Yaskawa INFORM job: SKRZYNIA_5440_90_STOPNI_20BR.JBI

/JOB
//NAME SKRZYNIA_5440_90_STOPNI_20BR
///FOLDERNAME 02-SKRZYNIE_JOBS
//POS
///NPOS 570,570,0,41,0,0
///TOOL 0
///POSTYPE PULSE
///PULSE
C00000=0,-52280,40443,0,6876,0
C00001=82314,-24956,17040,59626,-27382,6248
C00002=93910,-8625,17040,59626,-43355,6248
C00003=98846,-1061,-42166,80308,-57081,-16120
C00004=100452,6057,-48127,85711,-56704,-21322
C00005=95573,33077,-33257,84645,-64023,-26851
C00006=94102,33899,-31937,85246,-63371,-26689
C00007=95573,33077,-33257,84645,-64023,-26851
C00008=94862,31071,-36438,85313,-63677,-27192
C00009=95573,33077,-33257,84645,-64023,-26851
C00010=95263,33142,-33256,84677,-63995,-26850
C00011=95263,33142,-33256,84677,-63995,-26850
C00012=94017,33843,-32133,85187,-63445,-26710
C00013=95263,33142,-33256,84677,-63995,-26850
C00014=94657,31439,-35966,85248,-63701,-27141
C00015=95263,33142,-33256,84677,-63995,-26850
C00016=95260,33144,-33256,84678,-63995,-26850
C00017=95260,33144,-33256,84678,-63995,-26850
C00018=94022,33838,-32141,85183,-63448,-26711
C00019=95260,33144,-33256,84678,-63995,-26850
C00020=94618,31343,-36117,85281,-63684,-27157
C00021=95260,33144,-33256,84678,-63995,-26850
C00022=95258,25631,32269,66559,-75499,-2416
C00023=95258,25631,32269,66559,-75499,-2416
C00024=94181,26497,33533,66410,-74896,-2191
C00025=95658,30184,39035,66708,-78559,-2356
C00026=95217,30377,39331,66881,-79841,-2558
C00027=95258,25631,32269,66559,-75499,-2416
C00028=98811,21047,-15512,99242,-81394,-20987
C00029=98811,21047,-15512,99242,-81394,-20987
C00030=97775,21639,-14693,99563,-80753,-20993
C00031=98811,21047,-15512,99242,-81394,-20987
C00032=98206,18840,-18520,99489,-81124,-21211
C00033=98811,21047,-15512,99242,-81394,-20987
C00034=98765,34858,63506,90961,-74847,-417
C00035=98765,34858,63506,90961,-74847,-417
C00036=97741,35895,65220,90657,-74158,-246
C00037=98765,34858,63506,90961,-74847,-417
C00038=98337,32226,59232,91111,-74633,-884
C00039=98765,34858,63506,90961,-74847,-417
C00040=98728,21792,17445,103800,-78809,-12049
C00041=97232,27021,37502,101932,-75086,-7690
C00042=96358,27701,38514,101868,-74464,-7680
C00043=97232,27021,37502,101932,-75086,-7690
C00044=96733,24820,34282,102049,-74905,-7989
C00045=97232,27021,37502,101932,-75086,-7690
C00046=94428,854,16076,89248,-50738,-4740
C00047=88080,-20128,-3199,80943,-31244,-2335
C00048=48287,-44591,-17414,16172,-14532,25809
C00049=48287,-44591,-17414,16172,-14532,25809
C00050=86232,-22530,-5035,79517,-30097,-1713
C00051=97395,20012,29210,69700,-74457,-9077
C00052=97055,28839,36684,71776,-79389,-10554
C00053=97055,28839,36684,71776,-79389,-10554
C00054=96058,29646,37897,71666,-78799,-10362
C00055=97055,28839,36684,71776,-79389,-10554
C00056=96570,26659,33451,71832,-78911,-10777
C00057=97055,28839,36684,71776,-79389,-10554
C00058=99123,23256,18377,81563,-78104,3156
C00059=99123,23256,18377,81563,-78104,3156
C00060=98123,23909,19300,81582,-77442,3256
C00061=99123,23256,18377,81563,-78104,3156
C00062=98765,21723,16234,81638,-77830,3017
C00063=99123,23256,18377,81563,-78104,3156
C00064=99222,23346,17795,82202,-78388,4176
C00065=99222,23346,17795,82202,-78388,4176
C00066=98149,24045,18779,82229,-77677,4281
C00067=99222,23346,17795,82202,-78388,4176
C00068=98861,21801,15633,82278,-78114,4033
C00069=99222,23346,17795,82202,-78388,4176
C00070=101181,20053,13227,82362,-77850,3884
C00071=98477,12630,5837,99042,-72451,1602
C00072=98699,20516,16868,97574,-77073,2916
C00073=97285,21426,18123,97638,-76093,2915
C00074=98699,20516,16868,97574,-77073,2916
C00075=98338,19050,14867,97654,-76881,2766
C00076=98699,20516,16868,97574,-77073,2916
C00077=100004,19406,13931,91923,-76989,3541
C00078=99329,-2479,-35949,113241,-72472,-2557
C00079=60067,-64368,-72505,144806,-26050,-19168
C00080=60067,-50244,-32501,110603,-14199,-2207
C00081=63330,-26972,24478,18707,-56801,31483
C00082=87404,-10792,18065,42799,-49272,19535
C00083=97387,10585,22601,68146,-67072,4966
C00084=97468,27299,36957,71364,-78144,1860
C00085=96326,28190,38285,71210,-77468,2075
C00086=97482,27286,36940,71366,-78155,1858
C00087=97039,25308,34039,71414,-77723,1669
C00088=97482,27286,36940,71366,-78155,1858
C00089=99359,23449,25979,91431,-77368,-3620
C00090=98281,24164,26997,91405,-76622,-3568
C00091=99359,23449,25979,91431,-77368,-3620
C00092=98971,21749,23585,91505,-77132,-3802
C00093=99359,23449,25979,91431,-77368,-3620
C00094=96616,4564,7202,89178,-62130,-2525
C00095=94710,-18885,-12427,84555,-44606,134
C00096=42754,-66126,12236,-1301,3231,7194
C00097=0,-52280,40443,0,6876,0
C00098=0,-52280,40443,0,6876,0
C00099=48041,-29633,723,44271,-15597,-57965
C00100=48041,-29633,723,44271,-15597,-57965
C00101=55649,-15396,14646,74799,-19245,-69915
C00102=54283,-14162,15682,74499,-18354,-69938
C00103=56054,-13547,16209,75912,-19428,-70417
C00104=55649,-15396,14646,74799,-19245,-69915
C00105=51081,-17733,11598,53117,-16128,-61899
C00106=49703,-16390,12674,51759,-15261,-61403
C00107=50366,-16427,12642,52774,-15606,-61824
C00108=49536,-18455,11034,50297,-15435,-60714
C00109=50509,-19000,10610,51503,-15997,-61182
C00110=50873,-17966,11417,52677,-16048,-61710
C00111=49459,-16590,12517,51258,-15158,-61190
C00112=50592,-16429,12648,53120,-15720,-61960
C00113=50873,-17966,11417,52677,-16048,-61710
C00114=50703,-18403,11066,52155,-16024,-61477
C00115=50703,-18403,11066,52155,-16024,-61477
C00116=49026,-16768,12358,50435,-14971,-60844
C00117=50653,-16371,12680,53228,-15754,-62008
C00118=50703,-18403,11066,52155,-16024,-61477
C00119=50704,-18401,11069,52157,-16021,-61478
C00120=50704,-20525,5414,58956,-14779,-64789
C00121=49025,-18889,6668,57745,-13658,-64384
C00122=50799,-18420,7036,60610,-14610,-65581
C00123=50704,-20525,5414,58956,-14779,-64789
C00124=51005,-17995,11387,52847,-16122,-61778
C00125=51005,-17995,11387,52847,-16122,-61778
C00126=49564,-16598,12501,51417,-15218,-61257
C00127=50954,-16306,12737,53719,-15902,-62212
C00128=51005,-17995,11387,52847,-16122,-61778
C00129=51030,-17981,11395,52891,-16138,-61796
C00130=51030,-17981,11395,52891,-16138,-61796
C00131=49401,-16396,12662,51265,-15114,-61201
C00132=50908,-16047,12947,53789,-15850,-62250
C00133=51030,-17981,11395,52891,-16138,-61796
C00134=50945,-18019,11363,52741,-16103,-61737
C00135=50945,-16980,14081,49884,-16761,-60338
C00136=49117,-15186,15539,47848,-15653,-59576
C00137=50939,-14679,15960,50992,-16487,-60881
C00138=50945,-18019,11363,52741,-16103,-61737
C00139=50945,-18019,11363,52741,-16103,-61737
C00140=50945,-18556,9943,54337,-15776,-62517
C00141=48967,-16606,11493,52445,-14510,-61829
C00142=51083,-15952,12027,56053,-15559,-63336
C00143=50945,-18556,9943,54337,-15776,-62517
C00144=50945,-18019,11363,52741,-16103,-61737
C00145=51350,-15183,18375,46705,-17991,-58719
C00146=49319,-13187,20053,44263,-16830,-57796
C00147=51236,-12618,20544,47529,-17647,-59142
C00148=51350,-15183,18375,46705,-17991,-58719
C00149=50028,-23690,-6096,22921,-31075,-54538
C00150=50670,-23735,-6923,24003,-30760,-55076
C00151=48518,-21492,-5254,21861,-29696,-54082
C00152=50138,-21068,-4928,23831,-30039,-55022
C00153=50670,-23735,-6923,24003,-30760,-55076
C00154=49763,-24225,-29961,22080,-30065,-59113
C00155=49763,-24225,-29961,22080,-30065,-59113
C00156=47727,-21550,-27874,20313,-29013,-58119
C00157=49271,-21042,-27466,22016,-29310,-59069
C00158=49763,-24225,-29961,22080,-30065,-59113
C00159=50713,-12366,-58367,41124,-17813,-74400
C00160=50713,-12366,-58367,41124,-17813,-74400
C00161=48934,-9522,-55687,39981,-16902,-73526
C00162=50242,-8975,-55157,41389,-17374,-74448
C00163=50713,-12366,-58367,41124,-17813,-74400
C00164=50713,-12366,-58367,41124,-17813,-74400
C00165=50713,-12366,-58367,41124,-17813,-74400
C00166=48934,-9522,-55687,39981,-16902,-73526
C00167=50242,-8975,-55157,41389,-17374,-74448
C00168=50713,-12366,-58367,41124,-17813,-74400
C00169=49763,-25421,-36239,24565,-26935,-60445
C00170=43547,-31626,-19626,5157,-49140,-52118
C00171=40154,-51179,-915,24203,-8234,-36524
C00172=0,-52280,40443,0,6876,0
C00173=0,-52280,40443,0,6876,0
C00174=2117,-50103,-33543,4117,45077,-85249
C00175=-26439,-48928,-33543,4117,-52362,-85249
C00176=-1453,-29933,-32011,46693,-66666,-90474
C00177=24798,-19255,-10490,69050,-85424,-90395
C00178=18386,-22028,-12683,68302,-81515,-89477
///LIMIT ON
C00179=9843,-31743,-57176,61611,-65235,-99401
C00180=-39603,-23393,-71448,91573,-31907,-107123
C00181=-35705,5077,-63140,100511,-35979,-118164
C00182=-33789,12193,-59259,102607,-37482,-119984
C00183=-34998,13124,-58049,103267,-36945,-119997
C00184=-34401,14597,-56112,102586,-37131,-119778
C00185=-34998,13124,-58049,103267,-36945,-119997
C00186=-36388,13885,-57049,104079,-36338,-120048
C00187=-34998,13124,-58049,103267,-36945,-119997
C00188=-34008,-7969,-75285,118537,-50852,-116988
C00189=-26318,8527,-57077,128458,-81874,-108613
///LIMIT OFF
C00190=-23139,-1795,-12064,73373,-53703,-87448
C00191=-27830,-667,-10848,73187,-50621,-86997
C00192=-27373,916,-9115,73207,-50922,-87041
C00193=-27830,-667,-10848,73187,-50621,-86997
C00194=-28901,-207,-10348,73132,-49918,-86888
C00195=-27830,-667,-10848,73187,-50621,-86997
C00196=-37166,8347,13175,41366,-53536,-76331
C00197=-37403,7707,12401,41298,-53388,-76282
C00198=-36830,9273,14303,41455,-53750,-76396
C00199=-37403,7707,12401,41298,-53388,-76282
C00200=-38235,8246,13056,40951,-53040,-76025
C00201=-37403,7707,12401,41298,-53388,-76282
C00202=-30063,5992,18551,55847,-56234,-77619
C00203=-30754,7414,19761,55747,-55713,-77591
C00204=-30376,8670,21285,55817,-55984,-77619
C00205=-30754,7414,19761,55747,-55713,-77591
C00206=-31265,7672,20073,55566,-55435,-77478
C00207=-30085,6037,18588,55845,-56218,-77619
C00208=-25385,-1715,-9470,94765,-53990,-89712
C00209=-25885,-764,-8323,94779,-53645,-89697
C00210=-25564,418,-7032,94741,-53861,-89683
C00211=-25885,-764,-8323,94779,-53645,-89697
C00212=-26741,-428,-7957,94890,-53068,-89741
C00213=-25421,-1648,-9389,94767,-53966,-89710
C00214=-17789,-39335,-40320,90232,-41783,-86178
C00215=-25885,-761,-8324,94780,-53645,-89696
C00216=-25885,-761,-8324,94780,-53645,-89696
C00217=-25612,239,-7230,94748,-53828,-89684
C00218=-25885,-761,-8324,94780,-53645,-89696
C00219=-26712,-436,-7972,94885,-53087,-89742
C00220=-25885,-761,-8324,94780,-53645,-89696
C00221=-26038,-1317,-8919,94796,-53541,-89701
C00222=-18430,-29121,-33898,93348,-44706,-88207
C00223=-3209,-48313,-44409,84985,-37126,-83197
C00224=-3617,-53456,-46461,81793,-37023,-81323
C00225=-28991,-22310,-29554,94749,-46554,-89251
C00226=-30664,-6343,-14094,96248,-45630,-90223
C00227=-30664,-6343,-14094,96248,-45630,-90223
C00228=-30207,-5031,-12762,96238,-45949,-90236
C00229=-30664,-6343,-14094,96248,-45630,-90223
C00230=-31510,-5971,-13720,96406,-45066,-90297
C00231=-29506,-9179,-17232,96085,-46411,-90159
C00232=-30003,-8487,-16482,96169,-46079,-90194
C00233=-30881,-6301,-14053,96286,-45485,-90239
C00234=-30407,-4956,-12684,96275,-45813,-90252
C00235=-30881,-6301,-14053,96286,-45485,-90239
C00236=-31646,-5963,-13712,96429,-44974,-90305
C00237=-29893,-8752,-16772,96152,-46152,-90188
C00238=-30350,-7636,-15544,96220,-45845,-90215
C00239=-30881,-6301,-14053,96286,-45485,-90239
C00240=-30396,-4924,-12652,96275,-45822,-90251
C00241=-30881,-6301,-14053,96286,-45485,-90239
C00242=-31665,-5954,-13703,96434,-44961,-90308
C00243=-29959,-8593,-16598,96162,-46108,-90192
C00244=-26558,-19284,-27675,95285,-48332,-89713
C00245=-5136,-57382,-50746,80999,-31115,-81799
C00246=-5136,-57382,-50746,80999,-31115,-81799
C00247=-22762,-12288,-20025,94001,-55646,-89200
C00248=-24763,-3131,-11201,94769,-54426,-89746
C00249=-26203,-419,-7954,94818,-53430,-89712
C00250=-25939,548,-6896,94784,-53609,-89698
C00251=-26203,-419,-7954,94818,-53430,-89712
C00252=-26818,-174,-7689,94897,-53016,-89744
C00253=-24998,-2701,-10694,94780,-54264,-89743
C00254=-23275,-722,28392,94611,-50650,-77911
C00255=-21733,-16242,25206,75334,-39210,-63099
C00256=0,-52280,40443,0,6876,0
C00257=0,-52280,40443,0,6876,0
C00258=82314,-24956,17040,59626,-27382,6248
C00259=93910,-8625,17040,59626,-43355,6248
C00260=98846,-1061,-42166,80308,-57081,-16120
C00261=100452,6057,-48127,85711,-56704,-21322
C00262=95564,34698,-34234,85516,-63941,-27819
C00263=93687,36612,-31081,84292,-64733,-27467
C00264=93711,36598,-31105,84282,-64744,-27471
C00265=95564,34698,-34234,85516,-63941,-27819
C00266=96930,32282,-32252,82595,-65816,-26305
C00267=93663,32611,-31732,84127,-64318,-26195
C00268=93663,32611,-31732,84127,-64318,-26195
C00269=96930,32282,-32252,82595,-65816,-26305
C00270=96528,-7533,-34932,76119,-53878,-10439
C00271=88377,-34186,-45291,67238,-52212,-2442
C00272=73560,-62084,7826,28695,-34737,3666
C00273=0,-52280,40443,0,6876,0
C00274=0,-52280,40443,0,6876,0
C00275=2117,-50103,-33543,4117,45077,-85249
C00276=-26439,-48928,-33543,4117,-52362,-85249
C00277=-26439,-27355,-33543,41485,-52362,-85249
C00278=-39218,-24492,-41653,51934,-39374,-86964
C00279=-37997,-10433,-19136,70610,-34172,-88069
C00280=-38397,-8978,-17736,70703,-33874,-88109
C00281=-39218,-24492,-41653,51934,-39374,-86964
C00282=-26439,-27355,-33543,41485,-52362,-85249
C00283=1598,-24403,-16502,45671,-72599,-88798
C00284=-11365,-15171,10010,30164,-77975,-82960
C00285=-38112,4197,-14374,43778,-42973,-90436
C00286=-39116,7904,-10019,43942,-43580,-90646
C00287=-38495,8531,-9262,44482,-44499,-91194
C00288=-38112,4197,-14374,43778,-42973,-90436
C00289=-53220,-12364,-8957,19277,-47766,-73858
C00290=-11365,-15171,10010,30164,-77975,-82960
C00291=-16156,-38280,11293,23671,-42998,-42040
C00292=-11365,-47379,10010,30164,3063,-681
C00293=0,-52280,40443,0,6876,0
C00294=0,-36700,24612,-42871,-31823,-33862
C00295=44403,-30110,7154,24155,-23805,-45557
C00296=51347,-17798,16373,37641,-23556,-51399
C00297=51570,-17239,16856,38066,-23574,-51584
C00298=66153,-16343,3873,86567,-32078,-80939
C00299=60867,-15143,12446,70239,-26750,-71065
C00300=40431,-28773,9158,17648,-23273,-42875
C00301=0,-36700,24612,-42871,-31823,-33862
C00302=0,-52280,40443,0,6876,0
C00303=0,-52280,40443,0,6876,0
C00304=73560,-62084,7826,28695,-34737,3666
C00305=88377,-34186,-45291,67238,-52212,-2442
C00306=96528,-7533,-34932,76119,-53878,-10439
C00307=100432,21324,12575,83706,-77956,-7498
C00308=100432,21324,12575,83706,-77956,-7498
C00309=97224,21170,12361,83970,-75786,-7447
C00310=97224,21170,12361,83970,-75786,-7447
C00311=100432,21324,12575,83706,-77956,-7498
C00312=100432,21324,12575,83706,-77956,-7498
C00313=97481,25108,17890,83512,-78432,-7131
C00314=97624,25049,17805,83504,-78528,-7141
C00315=100432,21324,12575,83706,-77956,-7498
C00316=97137,1790,-11103,86179,-63102,-7963
C00317=99183,2264,5333,86781,-62651,-3264
C00318=99868,-33,22146,72719,-59601,5126
C00319=99028,-10516,17309,71061,-60695,4227
C00320=58820,-39124,10926,53325,-41870,3759
C00321=0,-52280,40443,0,6876,0
C00322=37281,-50778,-9546,79570,-75313,-71156
C00323=21038,-23698,-30323,82948,-81132,-85647
C00324=-27256,-5882,-14331,85818,-48304,-85968
C00325=-24751,2890,-4920,85349,-55822,-86178
C00326=-24793,2953,-4845,85351,-55796,-86173
C00327=-27256,-5882,-14331,85818,-48304,-85968
C00328=-21143,-15675,-23596,84785,-52496,-85466
C00329=35274,-15248,-23220,82440,-90817,-86704
C00330=35274,-15248,-23220,82440,-90817,-86704
C00331=-45551,161,-18089,35087,-36064,-73293
C00332=-42435,6767,-10562,40540,-41185,-77662
C00333=-42821,6494,-10882,40094,-40673,-77276
C00334=-45551,161,-18089,35087,-36064,-73293
C00335=-32891,-7184,-22739,69075,-41395,-83248
C00336=-29265,-39765,-39402,58096,-43152,-73226
C00337=-37287,-55159,35520,2191,5667,-2084
C00338=0,-52280,40443,0,6876,0
C00339=0,-36700,24612,-42871,-31823,-33862
C00340=44403,-30110,7154,24155,-23805,-45557
C00341=44403,-30110,7154,24155,-23805,-45557
C00342=42101,-12213,25656,103795,-5192,-78630
C00343=46259,-8171,27719,110365,-8144,-81138
C00344=67586,1814,51509,59543,-39517,-55403
C00345=68208,2417,52201,59959,-39833,-55512
C00346=58212,6581,49899,104854,-22273,-73944
C00347=50677,-23266,8367,38735,-22212,-52049
C00348=47073,-34549,9488,27883,-30316,-51458
C00349=0,-52280,40443,0,6876,0
C00350=0,-52280,40443,0,6876,0
C00351=73560,-62084,7826,28695,-34737,3666
C00352=96983,-27116,-23481,78724,-62297,-1998
C00353=100467,-7393,-15195,81625,-60158,-6002
C00354=99336,18440,8642,84276,-74234,-7647
C00355=99336,18440,8642,84276,-74234,-7647
C00356=97735,24994,14595,85350,-78994,-5109
C00357=97744,25074,13580,86004,-79195,-4385
C00358=99336,18440,8642,84276,-74234,-7647
C00359=99336,18440,8642,84276,-74234,-7647
C00360=97891,23737,8261,88167,-79183,-2386
C00361=97851,23541,8142,88101,-79081,-2507
C00362=99336,18440,8642,84276,-74234,-7647
C00363=99569,17008,9904,92397,-75404,-8157
C00364=97486,20835,7702,95706,-78487,-2828
C00365=97457,22481,19072,94521,-77544,253
C00366=101189,16995,13078,91997,-75892,-7124
C00367=89817,-14892,-20468,86994,-44415,-5457
C00368=100347,-21961,-42251,93939,-52125,-11121
C00369=60204,-59872,-73451,117647,-17639,-18840
C00370=37721,-67612,11381,1325,-438,7850
C00371=-37287,-55159,35520,2191,5667,-2084
C00372=-40042,-68802,-18337,47708,-19461,-45384
C00373=-28646,-23138,-32952,89786,-42552,-85395
C00374=-38882,-16596,-17625,44304,-41043,-72768
C00375=-42680,-6319,-12818,46127,-36112,-73823
C00376=-37459,704,-5408,52536,-43357,-78192
C00377=-32778,4349,-7465,59128,-48375,-83352
C00378=-42680,-6319,-12818,46127,-36112,-73823
C00379=-38882,-16596,-17625,44304,-41043,-72768
C00380=-28646,-23138,-32952,89786,-42552,-85395
C00381=-29905,-15291,-26411,91102,-43435,-86304
C00382=-25469,1350,-9790,89991,-54827,-86555
C00383=-24242,3379,-7505,89554,-57286,-86471
C00384=-29905,-15291,-26411,91102,-43435,-86304
C00385=-40042,-68802,-18337,47708,-19461,-45384
C00386=-37287,-55159,35520,2191,5667,-2084
C00387=0,-52280,40443,0,6876,0
C00388=37164,-60659,6466,13301,-5027,-19773
C00389=45362,-39990,2831,27538,-17767,-40935
C00390=57189,-26834,-7130,38780,-31731,-51561
C00391=63456,-14144,8594,45591,-40850,-50620
C00392=63325,-23790,-40688,66082,-30913,-63285
C00393=57189,-26834,-7130,38780,-31731,-51561
C00394=41180,-61187,4729,17280,-8498,-23442
C00395=0,-52280,40443,0,6876,0
C00396=37721,-67612,11381,1325,-438,7850
C00397=43180,-50572,-20637,6552,-29302,38834
C00398=79425,-37128,-15462,51820,-35721,18807
C00399=93702,-21743,-5664,65079,-41536,12324
C00400=94876,-11469,-23586,124528,-59237,-5423
C00401=92578,22421,15997,116595,-76671,1441
C00402=90287,21612,15190,116916,-75301,1087
C00403=91032,29854,33392,114957,-76206,4791
C00404=92578,22421,15997,116595,-76671,1441
C00405=94876,-11469,-23586,124528,-59237,-5423
C00406=93702,-22946,-9336,66730,-40927,11282
C00407=92743,-25622,-14104,67700,-39874,10604
C00408=95618,-29588,-12765,65168,-50072,21743
C00409=-36913,-32963,-979,75363,-26772,-58744
C00410=-42264,1508,8544,35869,-47237,-69477
C00411=-43183,4597,12058,35318,-46938,-69128
C00412=-43183,5775,16318,34276,-48598,-68388
C00413=-42264,1508,8544,35869,-47237,-69477
C00414=41438,-37635,17580,13151,-29920,-38779
C00415=54964,-26842,8528,44141,-23181,-52038
C00416=50761,-21373,7883,46957,-18149,-54038
C00417=65214,-17346,-4869,103105,-32325,-89305
C00418=65312,-6152,27526,81270,-31139,-77237
C00419=56762,-20631,11812,69834,-24329,-69917
C00420=46096,-45842,-2681,20981,-19497,-36310
C00421=41180,-61187,4729,17280,-8498,-23442
C00422=0,-52280,40443,0,6876,0
C00423=0,-52280,40443,0,6876,0
C00424=37721,-67612,11381,1325,-438,7850
C00425=43180,-50572,-20637,6552,-29302,38834
C00426=79425,-37128,-15462,51820,-35721,18807
C00427=90367,-20498,-14913,71355,-37589,8070
C00428=98864,-2001,-14672,90389,-62789,-3799
C00429=98767,21176,13691,87588,-77304,-2577
C00430=98123,23617,17097,87345,-78645,-2335
C00431=97979,23711,17231,87352,-78549,-2326
C00432=98864,-2001,-14672,90389,-62789,-3799
C00433=100472,-329,-13432,98539,-67097,-6304
C00434=92822,-26306,-37175,103295,-43881,-7703
C00435=68601,-52593,-52127,95725,-25602,-3235
C00436=80632,-38079,-20908,64053,-45216,12949
C00437=43180,-50572,-20637,6552,-29302,38834
C00438=37721,-67612,11381,1325,-438,7850
C00439=0,-52280,40443,0,6876,0
C00440=0,-52280,40443,0,6876,0
C00441=0,-52280,40443,0,-39412,36675
C00442=-54026,-30203,28811,-7745,-28969,-5087
C00443=-30389,-9386,-5824,79667,-43789,-73484
C00444=-32979,-3325,255,79720,-41988,-73575
C00445=-25304,6223,10893,81656,-55729,-74481
C00446=-23842,8927,14147,81883,-58875,-74544
C00447=-30389,-9386,-5824,79667,-43789,-73484
C00448=-32145,-6440,-2937,79673,-42575,-73527
C00449=-25014,6414,11121,81706,-56254,-74506
C00450=-23603,11547,23533,79434,-59735,-72187
C00451=-32145,-5050,2357,77009,-42992,-71800
C00452=-35251,-18143,20376,53513,-41117,-59413
C00453=-9534,-43450,13514,26959,-29486,-38723
C00454=-22834,-59963,22946,6692,-2150,-9612
C00455=0,-52280,40443,0,6876,0
C00456=23708,-46776,23536,16027,-4787,-19738
C00457=50917,-40459,4132,34421,-18173,-42391
C00458=51059,-36587,4608,36647,-19418,-45358
C00459=50113,-22729,10834,36393,-23396,-50963
C00460=62046,-17757,4067,79440,-27252,-76630
C00461=63804,-15651,7512,80030,-29507,-77065
C00462=50113,-22729,10834,36393,-23396,-50963
C00463=31287,-69981,-10850,7253,-6843,-20996
C00464=19644,-57271,30737,863,5243,-2499
C00465=0,-52280,40443,0,6876,0
C00466=0,-52280,40443,0,6876,0
C00467=37721,-67612,11381,1325,-438,7850
C00468=43180,-50572,-20637,6552,-29302,38834
C00469=90700,-21740,-5659,63738,-39702,12884
C00470=98442,-3149,-15680,86092,-59018,-2413
C00471=96855,-5742,-18360,86176,-57949,-2343
C00472=99185,22470,15697,83135,-77937,-1734
C00473=97717,21807,14770,83256,-76932,-1762
C00474=97717,21807,14770,83256,-76932,-1762
C00475=99185,24652,26607,82087,-78431,1026
C00476=99185,22470,15697,83135,-77937,-1734
C00477=97852,24994,19264,82957,-78889,-1504
C00478=97683,25109,19429,82963,-78778,-1488
C00479=99870,24121,23963,82328,-78767,341
C00480=99670,26545,33629,93870,-78468,540
C00481=97522,25636,31977,94228,-76846,981
C00482=97561,29801,46317,92820,-76116,4162
C00483=100647,24287,31478,94135,-78005,1371
C00484=100690,13539,3274,89268,-73991,-3693
C00485=95827,-6765,-19867,92747,-56076,-4624
C00486=92822,-26306,-37175,103295,-43881,-7703
C00487=68601,-52593,-52127,95725,-25602,-3235
C00488=80632,-38079,-20908,64053,-45216,12949
C00489=43180,-50572,-20637,6552,-29302,38834
C00490=37721,-67612,11381,1325,-438,7850
C00491=0,-52280,40443,0,6876,0
C00492=0,-52280,40443,0,6876,0
C00493=0,-52280,40443,0,-39412,36675
C00494=-54026,-30203,28811,-7745,-28969,-5087
C00495=-81492,-18979,22896,-11682,-23662,-26316
C00496=-32145,-2720,10458,73217,-43826,-69319
C00497=-32145,-2720,10458,73217,-43826,-69319
C00498=-25800,12961,35355,74076,-56913,-68018
C00499=-23961,12723,28512,77913,-59573,-70804
C00500=-32145,-2720,10458,73217,-43826,-69319
C00501=-34274,-9754,-24316,117159,-46217,-86271
C00502=-34274,-9754,-24316,117159,-46217,-86271
C00503=-29822,-1437,-15851,112752,-53901,-84078
C00504=-28945,-336,-14662,112011,-55335,-83695
C00505=-34274,-9754,-24316,117159,-46217,-86271
C00506=-34422,-9999,20796,72411,-42519,-66994
C00507=-35251,-18143,20376,53513,-41117,-59413
C00508=-9534,-43450,13514,26959,-29486,-38723
C00509=-22834,-59963,22946,6692,-2150,-9612
C00510=0,-52280,40443,0,6876,0
C00511=44101,-76445,-48847,15697,-17168,-40457
C00512=49121,-28282,-35458,21895,-29219,-59001
C00513=50484,-13386,-55713,36158,-19724,-71897
C00514=55938,-10187,-55661,55618,-22248,-82832
C00515=57262,15098,-57515,78189,-20957,-89981
C00516=57264,15099,-57513,78187,-20957,-89981
C00517=50484,-13386,-55713,36158,-19724,-71897
C00518=49763,-25421,-36239,24565,-26935,-60445
C00519=50529,-22709,-3778,22940,-31995,-54502
C00520=45389,-28224,4312,35967,-15579,-54278
C00521=40154,-51179,-915,24203,-8234,-36524
C00522=0,-52280,40443,0,6876,0
C00523=0,-52280,40443,0,6876,0
C00524=37721,-67612,11381,1325,-438,7850
C00525=43181,-50571,-20637,6551,-29300,38834
C00526=87798,-21399,-8795,65098,-36955,11822
C00527=85232,-2754,25377,50981,-49542,17626
C00528=95618,10017,30418,66150,-65403,10402
C00529=98328,26728,37723,75385,-78922,5377
C00530=97988,24882,21615,85608,-78767,-653
C00531=97988,24882,21615,85608,-78767,-653
C00532=97883,29022,44703,72741,-79810,7156
C00533=99206,10365,20042,80584,-66974,4673
C00534=97521,29471,41231,76536,-79243,4998
C00535=96632,30112,41879,71718,-79572,5847
C00536=99876,18242,24023,78306,-74179,3477
C00537=99266,24955,27205,94359,-77696,-2486
C00538=97755,22340,21286,94814,-76951,-3534
C00539=97755,24574,30760,93819,-76338,-1256
C00540=99407,24851,31160,93832,-77451,-1162
C00541=97945,29512,41217,93178,-77856,493
C00542=97945,34878,57710,91784,-77173,3936
C00543=99407,24851,31160,93832,-77451,-1162
C00544=97855,1258,8902,87977,-59100,1980
C00545=95777,-4741,32780,63689,-53673,17098
C00546=72477,-33752,-3372,52810,-39669,19964
C00547=0,-52278,40443,0,6872,5
C00548=0,-52278,40443,31822,-65283,-46097
C00549=-7820,3000,44222,77356,-66876,-70486
C00550=-24244,23423,72059,64993,-61079,-67138
C00551=-27261,30732,84230,62108,-60720,-65392
C00552=-22394,37028,87531,68934,-68535,-64461
C00553=-24244,23423,72059,64993,-61079,-67138
C00554=3014,-20441,-7349,104591,-68614,-79454
C00555=6322,-14118,13197,96169,-69167,-72790
C00556=14133,-16757,18528,88010,-59455,-67296
C00557=-10261,-46634,14475,36899,-22136,-31570
C00558=-22834,-59963,22946,6692,-2150,-9612
C00559=0,-52280,40443,0,6876,0
C00560=23708,-46776,23536,16027,-4787,-19738
C00561=50917,-40459,4132,34421,-18173,-42391
C00562=49876,-21948,7530,68838,-10324,-59148
C00563=46721,-18942,9765,68167,-8197,-59205
C00564=59102,-15651,-1637,118714,-27356,-88041
C00565=59185,-13834,7185,105143,-23914,-78054
C00566=45927,-22803,4403,78462,-8511,-64553
C00567=62498,-35400,-2607,72048,-19281,-59202
C00568=31287,-69981,-10850,7253,-6843,-20996
C00569=0,-52280,40443,0,6876,0
BC00000=487510
BC00001=445130
BC00002=445130
BC00003=445130
BC00004=445130
BC00005=468227
BC00006=468227
BC00007=468227
BC00008=468227
BC00009=468227
BC00010=514421
BC00011=514421
BC00012=514421
BC00013=514421
BC00014=514421
BC00015=514421
BC00016=560588
BC00017=560588
BC00018=560588
BC00019=560588
BC00020=560588
BC00021=560588
BC00022=536404
BC00023=536404
BC00024=536404
BC00025=536404
BC00026=536404
BC00027=536404
BC00028=582458
BC00029=582458
BC00030=582458
BC00031=582458
BC00032=582458
BC00033=582458
BC00034=581206
BC00035=581206
BC00036=581206
BC00037=581206
BC00038=581206
BC00039=581206
BC00040=626960
BC00041=626960
BC00042=626960
BC00043=626960
BC00044=626960
BC00045=626960
BC00046=604255
BC00047=604255
BC00048=604255
BC00049=734179
BC00050=734179
BC00051=772491
BC00052=770398
BC00053=770398
BC00054=770398
BC00055=770398
BC00056=770398
BC00057=770398
BC00058=820815
BC00059=820815
BC00060=820815
BC00061=820815
BC00062=820815
BC00063=820815
BC00064=866263
BC00065=866263
BC00066=866260
BC00067=866263
BC00068=866263
BC00069=866263
BC00070=866263
BC00071=903321
BC00072=903321
BC00073=903321
BC00074=903321
BC00075=903321
BC00076=903321
BC00077=881024
BC00078=869038
BC00079=872244
BC00080=872244
BC00081=964954
BC00082=968815
BC00083=986882
BC00084=986882
BC00085=986882
BC00086=986882
BC00087=986882
BC00088=986882
BC00089=1031858
BC00090=1031858
BC00091=1031858
BC00092=1031858
BC00093=1031858
BC00094=991476
BC00095=978789
BC00096=857759
BC00097=811793
BC00098=811793
BC00099=953382
BC00100=1007225
BC00101=1007225
BC00102=1007225
BC00103=1007225
BC00104=1007225
BC00105=953382
BC00106=953382
BC00107=953383
BC00108=953382
BC00109=888056
BC00110=888056
BC00111=888056
BC00112=888056
BC00113=888056
BC00114=830714
BC00115=830714
BC00116=830714
BC00117=830714
BC00118=830714
BC00119=764829
BC00120=764829
BC00121=764829
BC00122=764829
BC00123=764829
BC00124=707174
BC00125=707174
BC00126=707174
BC00127=707174
BC00128=707174
BC00129=642071
BC00130=642071
BC00131=642071
BC00132=642071
BC00133=642071
BC00134=584746
BC00135=584746
BC00136=584746
BC00137=584746
BC00138=584746
BC00139=519232
BC00140=519232
BC00141=519232
BC00142=519232
BC00143=519232
BC00144=461813
BC00145=461813
BC00146=461813
BC00147=461813
BC00148=461813
BC00149=459544
BC00150=459544
BC00151=459544
BC00152=459544
BC00153=459544
BC00154=459544
BC00155=459544
BC00156=459544
BC00157=459544
BC00158=459544
BC00159=459544
BC00160=459544
BC00161=459544
BC00162=459544
BC00163=459544
BC00164=413461
BC00165=413461
BC00166=413461
BC00167=413461
BC00168=413461
BC00169=459544
BC00170=462325
BC00171=533216
BC00172=533216
BC00173=492150
BC00174=423885
BC00175=423885
BC00176=519103
BC00177=542802
BC00178=634915
BC00179=493160
BC00180=493160
BC00181=517936
BC00182=517447
BC00183=516208
BC00184=516208
BC00185=516208
BC00186=516208
BC00187=516208
BC00188=525487
BC00189=485388
BC00190=500803
BC00191=500803
BC00192=500803
BC00193=500803
BC00194=500803
BC00195=500803
BC00196=585253
BC00197=585253
BC00198=585253
BC00199=585253
BC00200=585253
BC00201=585253
BC00202=600589
BC00203=600589
BC00204=600589
BC00205=600589
BC00206=600589
BC00207=600589
BC00208=646713
BC00209=646713
BC00210=646713
BC00211=646713
BC00212=646713
BC00213=646713
BC00214=659006
BC00215=692822
BC00216=692822
BC00217=692822
BC00218=692822
BC00219=692822
BC00220=692822
BC00221=669701
BC00222=669701
BC00223=669701
BC00224=791136
BC00225=762000
BC00226=762000
BC00227=762000
BC00228=762000
BC00229=762000
BC00230=762000
BC00231=762000
BC00232=831025
BC00233=831025
BC00234=831025
BC00235=831025
BC00236=831025
BC00237=831025
BC00238=877128
BC00239=877128
BC00240=877128
BC00241=877128
BC00242=877128
BC00243=877128
BC00244=854090
BC00245=854090
BC00246=990684
BC00247=992363
BC00248=992364
BC00249=992364
BC00250=992364
BC00251=992364
BC00252=992364
BC00253=992364
BC00254=941750
BC00255=932032
BC00256=834170
BC00257=445130
BC00258=445130
BC00259=445130
BC00260=445130
BC00261=445130
BC00262=475938
BC00263=475938
BC00264=468314
BC00265=475938
BC00266=515329
BC00267=515329
BC00268=507641
BC00269=515329
BC00270=542207
BC00271=542207
BC00272=542207
BC00273=542207
BC00274=492150
BC00275=423885
BC00276=423885
BC00277=423885
BC00278=423885
BC00279=406365
BC00280=406365
BC00281=423885
BC00282=423885
BC00283=423885
BC00284=423885
BC00285=507950
BC00286=507950
BC00287=500226
BC00288=507950
BC00289=493160
BC00290=493160
BC00291=493160
BC00292=493160
BC00293=493160
BC00294=582810
BC00295=655182
BC00296=712102
BC00297=712780
BC00298=712780
BC00299=769565
BC00300=773753
BC00301=582810
BC00302=493160
BC00303=542207
BC00304=542207
BC00305=542207
BC00306=590944
BC00307=543764
BC00308=459277
BC00309=459277
BC00310=451665
BC00311=459277
BC00312=520748
BC00313=520748
BC00314=528468
BC00315=520748
BC00316=524597
BC00317=604006
BC00318=584417
BC00319=584417
BC00320=584417
BC00321=584417
BC00322=542360
BC00323=521200
BC00324=474976
BC00325=474976
BC00326=482600
BC00327=474976
BC00328=474976
BC00329=474976
BC00330=630364
BC00331=628593
BC00332=624867
BC00333=617183
BC00334=631527
BC00335=617183
BC00336=617427
BC00337=620193
BC00338=620193
BC00339=812803
BC00340=887783
BC00341=927066
BC00342=893694
BC00343=914884
BC00344=936389
BC00345=992711
BC00346=992711
BC00347=962387
BC00348=853059
BC00349=542207
BC00350=542207
BC00351=542207
BC00352=541760
BC00353=590944
BC00354=571989
BC00355=566860
BC00356=566868
BC00357=574636
BC00358=566860
BC00359=635958
BC00360=635958
BC00361=643642
BC00362=635958
BC00363=664809
BC00364=664812
BC00365=664812
BC00366=664812
BC00367=635118
BC00368=635118
BC00369=656468
BC00370=665809
BC00371=620193
BC00372=620193
BC00373=635598
BC00374=635598
BC00375=635598
BC00376=635598
BC00377=635598
BC00378=635598
BC00379=635598
BC00380=635598
BC00381=658627
BC00382=658627
BC00383=666320
BC00384=658627
BC00385=620193
BC00386=620193
BC00387=620193
BC00388=561542
BC00389=498768
BC00390=452071
BC00391=452071
BC00392=454195
BC00393=452071
BC00394=524165
BC00395=524165
BC00396=733103
BC00397=733103
BC00398=615417
BC00399=615411
BC00400=615411
BC00401=615411
BC00402=615411
BC00403=615411
BC00404=615411
BC00405=615411
BC00406=615411
BC00407=615417
BC00408=615413
BC00409=696009
BC00410=735643
BC00411=735643
BC00412=739967
BC00413=735643
BC00414=549560
BC00415=580754
BC00416=589556
BC00417=589556
BC00418=626883
BC00419=634257
BC00420=536572
BC00421=561088
BC00422=547800
BC00423=733103
BC00424=733103
BC00425=733103
BC00426=754456
BC00427=776787
BC00428=740531
BC00429=740531
BC00430=740531
BC00431=748211
BC00432=740531
BC00433=750469
BC00434=750469
BC00435=750469
BC00436=783373
BC00437=795297
BC00438=733103
BC00439=733103
BC00440=672709
BC00441=672709
BC00442=762701
BC00443=743900
BC00444=736524
BC00445=736351
BC00446=743900
BC00447=743900
BC00448=759331
BC00449=759331
BC00450=759331
BC00451=759331
BC00452=750104
BC00453=672725
BC00454=672725
BC00455=672725
BC00456=766882
BC00457=791101
BC00458=802867
BC00459=836517
BC00460=836517
BC00461=895034
BC00462=836517
BC00463=618402
BC00464=618402
BC00465=618402
BC00466=733103
BC00467=733103
BC00468=828551
BC00469=828551
BC00470=815683
BC00471=817504
BC00472=817504
BC00473=817504
BC00474=825298
BC00475=817504
BC00476=863642
BC00477=863642
BC00478=871437
BC00479=863642
BC00480=893797
BC00481=893797
BC00482=893797
BC00483=893797
BC00484=885212
BC00485=863492
BC00486=830221
BC00487=811977
BC00488=783373
BC00489=795297
BC00490=733103
BC00491=733103
BC00492=672709
BC00493=672709
BC00494=762701
BC00495=791880
BC00496=819491
BC00497=819491
BC00498=817331
BC00499=817331
BC00500=817326
BC00501=863478
BC00502=863478
BC00503=863478
BC00504=871062
BC00505=863478
BC00506=774095
BC00507=750104
BC00508=672725
BC00509=672725
BC00510=672725
BC00511=528256
BC00512=459544
BC00513=459544
BC00514=458584
BC00515=459547
BC00516=450935
BC00517=459544
BC00518=459544
BC00519=459544
BC00520=459540
BC00521=533216
BC00522=533216
BC00523=733103
BC00524=733103
BC00525=976969
BC00526=974440
BC00527=928072
BC00528=935112
BC00529=947035
BC00530=947035
BC00531=954731
BC00532=947035
BC00533=969317
BC00534=979591
BC00535=979591
BC00536=979591
BC00537=1019602
BC00538=1019602
BC00539=1019602
BC00540=1019602
BC00541=1027651
BC00542=1027651
BC00543=1019602
BC00544=991903
BC00545=955597
BC00546=952322
BC00547=852584
BC00548=921533
BC00549=958534
BC00550=946591
BC00551=946591
BC00552=946592
BC00553=954904
BC00554=963295
BC00555=934184
BC00556=908449
BC00557=754884
BC00558=672725
BC00559=672725
BC00560=562340
BC00561=452362
BC00562=452362
BC00563=452362
BC00564=452362
BC00565=513216
BC00566=512110
BC00567=512008
BC00568=742282
BC00569=742282
///POSTYPE BASE
///RECTAN
///RCONF 1,0,0,0,0,0,0,0,0,0,0,0,0,0,0,0,0,0,0,0,0,0,0,0
P00006=0.000,0.000,0.000,0.0000,0.0000,0.0000
///RCONF 0,0,0,0,0,0,0,0,0,0,0,0,0,0,0,0,0,0,0,0,0,0,0,0
P00058=0.000,0.000,3.000,0.0000,0.0000,0.0000
///RCONF 1,0,0,0,0,0,0,0,0,0,0,0,0,0,0,0,0,0,0,0,0,0,0,0
P00300=-0.036,-1.505,2.318,0.0000,0.0000,0.0000
P00301=0.046,-2.112,7.779,0.0000,0.0000,0.0000
P00302=-0.180,-2.409,6.326,0.0000,0.0000,0.0000
///RCONF 0,0,0,0,0,0,0,0,0,0,0,0,0,0,0,0,0,0,0,0,0,0,0,0
P00303=-0.004,-1.437,-4.584,0.0000,0.0000,0.0000
P00304=0.028,-1.666,-4.234,0.0000,0.0000,0.0000
P00305=-0.003,-1.920,-3.501,0.0000,0.0000,0.0000
P00306=0.015,-2.252,-3.054,0.0000,0.0000,0.0000
P00307=0.019,-2.151,-5.077,0.0000,0.0000,0.0000
P00308=-0.003,-2.092,-4.888,0.0000,0.0000,0.0000
P00309=-0.040,-2.205,-4.992,0.0000,0.0000,0.0000
P00310=-0.006,-2.490,-5.925,0.0000,0.0000,0.0000
P00311=-0.007,-2.079,-5.307,0.0000,0.0000,0.0000
P00312=-0.032,2.202,-7.632,0.0000,0.0000,0.0000
///RCONF 1,0,0,0,0,0,0,0,0,0,0,0,0,0,0,0,0,0,0,0,0,0,0,0
P00349=0.060,0.167,-1.133,0.0000,0.0000,0.0000
///RCONF 0,0,0,0,0,0,0,0,0,0,0,0,0,0,0,0,0,0,0,0,0,0,0,0
P00350=11.519,-0.008,1.149,0.0000,0.0000,0.0000
P00351=13.563,-0.027,-0.653,0.0000,0.0000,0.0000
P00352=13.252,-0.027,-0.827,0.0000,0.0000,0.0000
P00353=10.971,-0.082,0.776,0.0000,0.0000,0.0000
P00354=-0.024,2.508,-1.824,0.0000,0.0000,0.0000
P00355=-0.001,2.528,-1.131,0.0000,0.0000,0.0000
P00356=-0.034,2.921,-0.262,0.0000,0.0000,0.0000
P00357=0.003,3.386,-0.091,0.0000,0.0000,0.0000
P00358=0.014,3.037,-0.020,0.0000,0.0000,0.0000
P00359=-0.005,2.731,0.912,0.0000,0.0000,0.0000
P00360=-0.011,3.412,0.438,0.0000,0.0000,0.0000
P00361=0.018,3.050,1.253,0.0000,0.0000,0.0000
P00362=0.014,2.784,0.148,0.0000,0.0000,0.0000
P00400=5.920,-3.503,-0.024,0.0000,0.0000,0.0000
P00401=3.430,-0.021,1.131,0.0000,0.0000,0.0000
P00402=-0.253,1.107,3.062,0.0000,0.0000,0.0000
P00403=-3.666,-0.015,5.328,0.0000,0.0000,0.0000
///RCONF 1,0,0,0,0,0,0,0,0,0,0,0,0,0,0,0,0,0,0,0,0,0,0,0
P00404=0.029,4.189,-1.030,0.0000,0.0000,0.0000
///RCONF 0,0,0,0,0,0,0,0,0,0,0,0,0,0,0,0,0,0,0,0,0,0,0,0
P00405=2.420,0.007,1.427,0.0000,0.0000,0.0000
P00406=3.513,-0.022,0.429,0.0000,0.0000,0.0000
///RCONF 1,0,0,0,1,0,0,0,0,0,0,0,0,0,0,0,0,0,0,0,0,0,0,0
P00407=-0.029,2.348,-1.469,0.0000,0.0000,0.0000
P00408=0.010,1.346,-1.479,0.0000,0.0000,0.0000
///RCONF 1,0,0,0,0,0,0,0,0,0,0,0,0,0,0,0,0,0,0,0,0,0,0,0
P00409=-0.026,2.090,-1.483,0.0000,0.0000,0.0000
P00410=0.001,4.491,-0.583,0.0000,0.0000,0.0000
///RCONF 1,0,0,0,1,0,0,0,0,0,0,0,0,0,0,0,0,0,0,0,0,0,0,0
P00411=-0.015,3.627,0.872,0.0000,0.0000,0.0000
//INST
///DATE 2024/10/02 15:26
///ATTR SC,RW
///GROUP1 RB1,BS1
NOP
CALL JOB:MOVE_INTO_TUNNEL
MOVJ C00000 BC00000 VJ=10.00
MOVJ C00001 BC00001 VJ=30.00
MOVJ C00002 BC00002 VJ=30.00
MOVL C00003 BC00003 V=500.0
MOVJ C00004 BC00004 VJ=30.00
'------------------------
'W65.3
'------------------------
MOVL C00005 BC00005 V=333.3 PL=0
REFP 3 C00006 BC00006
CALL JOB:SEARCH-R1
SET P0300 P0006
SFTON P0300
MOVL C00007 BC00007 V=333.3 PL=0
REFP 3 C00008 BC00008
CALL JOB:SEARCH-R1
SET P0300 P0006
SFTON P0300
MOVL C00009 BC00009 V=333.3 PL=0
SFTOF
'------------------------
'W65.5
'------------------------
MOVL C00010 BC00010 V=500.0
MOVL C00011 BC00011 V=333.3 PL=0
REFP 3 C00012 BC00012
CALL JOB:SEARCH-R1
SET P0301 P0006
SFTON P0301
MOVL C00013 BC00013 V=333.3 PL=0
REFP 3 C00014 BC00014
CALL JOB:SEARCH-R1
SET P0301 P0006
SFTON P0301
MOVL C00015 BC00015 V=333.3 PL=0
SFTOF
'------------------------
'W65.7
'------------------------
MOVL C00016 BC00016 V=500.0
MOVL C00017 BC00017 V=333.3 PL=0
REFP 3 C00018 BC00018
CALL JOB:SEARCH-R1
SET P0302 P0006
SFTON P0302
MOVL C00019 BC00019 V=333.3 PL=0
REFP 3 C00020 BC00020
CALL JOB:SEARCH-R1
SET P0302 P0006
SFTON P0302
MOVL C00021 BC00021 V=500.0 PL=0
SFTOF
'------------------------
'W65.10
'------------------------
MOVL C00022 BC00022 V=500.0
MOVL C00023 BC00023 V=333.3 PL=0
REFP 3 C00024 BC00024
CALL JOB:SEARCH-R1
SET P0303 P0006
SFTON P0303
MOVL C00025 BC00025 V=333.3 PL=0
REFP 3 C00026 BC00026
CALL JOB:SEARCH-R1
SET P0303 P0006
SFTON P0303
MOVL C00027 BC00027 V=333.3 PL=0
SFTOF
'------------------------
'W65.12
'------------------------
MOVL C00028 BC00028 V=500.0
MOVL C00029 BC00029 V=333.3 PL=0
REFP 3 C00030 BC00030
CALL JOB:SEARCH-R1
SET P0304 P0006
SFTON P0304
MOVL C00031 BC00031 V=333.3 PL=0
REFP 3 C00032 BC00032
CALL JOB:SEARCH-R1
SET P0304 P0006
SFTON P0304
MOVL C00033 BC00033 V=333.3 PL=0
SFTOF
'------------------------
'W65.15
'------------------------
MOVL C00034 BC00034 V=500.0
MOVL C00035 BC00035 V=333.3 PL=0
REFP 3 C00036 BC00036
CALL JOB:SEARCH-R1
SET P0305 P0006
SFTON P0305
MOVL C00037 BC00037 V=333.3 PL=0
REFP 3 C00038 BC00038
CALL JOB:SEARCH-R1
SET P0305 P0006
SFTON P0305
MOVL C00039 BC00039 V=333.3 PL=0
SFTOF
'------------------------
'W65.17
'------------------------
MOVL C00040 BC00040 V=500.0
MOVL C00041 BC00041 V=166.7 PL=0
REFP 3 C00042 BC00042
CALL JOB:SEARCH-R1
SET P0306 P0006
SFTON P0306
MOVL C00043 BC00043 V=333.3 PL=0
REFP 3 C00044 BC00044
CALL JOB:SEARCH-R1
SET P0306 P0006
SFTON P0306
MOVL C00045 BC00045 V=500.0 PL=0
SFTOF
MOVL C00046 BC00046 V=500.0
MOVL C00047 BC00047 V=500.0
MOVL C00048 BC00048 V=500.0
MOVJ C00049 BC00049 VJ=30.00
MOVL C00050 BC00050 V=500.0
MOVL C00051 BC00051 V=500.0
'------------------------
'W65.20
'------------------------
COMM MOVL C00052 BC00052 V=500.0
COMM MOVL C00053 BC00053 V=333.3 PL=0
COMM REFP 3 C00054 BC00054
COMM CALL JOB:SEARCH-R1
COMM SET P0307 P0006
COMM SFTON P0307
COMM MOVL C00055 BC00055 V=333.3 PL=0
COMM REFP 3 C00056 BC00056
COMM CALL JOB:SEARCH-R1
COMM SET P0307 P0006
COMM SFTON P0307
COMM MOVL C00057 BC00057 V=500.0 PL=0
COMM SFTOF
COMM '------------------------
COMM 'W65.23
'------------------------
MOVL C00058 BC00058 V=500.0
MOVL C00059 BC00059 V=333.3 PL=0
REFP 3 C00060 BC00060
CALL JOB:SEARCH-R1
SET P0308 P0006
SFTON P0308
MOVL C00061 BC00061 V=333.3 PL=0
REFP 3 C00062 BC00062
CALL JOB:SEARCH-R1
SET P0308 P0006
SFTON P0308
MOVL C00063 BC00063 V=500.0 PL=0
SFTOF
'------------------------
'W65.25
'------------------------
MOVL C00064 BC00064 V=500.0
MOVL C00065 BC00065 V=333.3 PL=0
REFP 3 C00066 BC00066
CALL JOB:SEARCH-R1
SET P0309 P0006
SFTON P0309
MOVL C00067 BC00067 V=333.3 PL=0
REFP 3 C00068 BC00068
CALL JOB:SEARCH-R1
SET P0309 P0006
SFTON P0309
MOVL C00069 BC00069 V=500.0 PL=0
SFTOF
MOVL C00070 BC00070 V=250.0
MOVL C00071 BC00071 V=416.7
MOVL C00072 BC00072 V=166.7
REFP 3 C00073 BC00073
CALL JOB:SEARCH-R1
SET P0310 P0006
SFTON P0310
MOVL C00074 BC00074 V=166.7 PL=0
REFP 3 C00075 BC00075
CALL JOB:SEARCH-R1
SET P0310 P0006
SFTON P0310
SFTOF
MOVL C00076 BC00076 V=333.3 PL=0
MOVL C00077 BC00077 V=500.0
MOVL C00078 BC00078 V=500.0
MOVL C00079 BC00079 V=500.0
MOVL C00080 BC00080 V=500.0
MOVL C00081 BC00081 V=250.0
MOVL C00082 BC00082 V=500.0
MOVL C00083 BC00083 V=500.0
'------------------------
'W65.28
'------------------------
MOVL C00084 BC00084 V=166.7 PL=0
REFP 3 C00085 BC00085
CALL JOB:SEARCH-R1
SET P0311 P0006
SFTON P0311
MOVL C00086 BC00086 V=166.7 PL=0
REFP 3 C00087 BC00087
CALL JOB:SEARCH-R1
SET P0311 P0006
SFTON P0311
MOVL C00088 BC00088 V=250.0 PL=0
SFTOF
'------------------------
'W65.30
'------------------------
MOVL C00089 BC00089 V=333.3 PL=0
REFP 3 C00090 BC00090
CALL JOB:SEARCH-R1
SET P0312 P0006
SFTON P0312
MOVL C00091 BC00091 V=333.3 PL=0
REFP 3 C00092 BC00092
CALL JOB:SEARCH-R1
SET P0312 P0006
SFTON P0312
MOVL C00093 BC00093 V=333.3 PL=0
SFTOF
MOVL C00094 BC00094 V=500.0
MOVL C00095 BC00095 V=500.0
MOVJ C00096 BC00096 VJ=30.00
MOVJ C00097 BC00097 VJ=30.00
MOVJ C00098 BC00098 VJ=30.00
MOVJ C00099 BC00099 VJ=30.00
MOVJ C00100 BC00100 VJ=50.00
MOVL C00101 BC00101 V=166.7 PL=0
REFP 3 C00102 BC00102
CALL JOB:SEARCH-R1
IMOV P0058 V=16.7
SET P0349 P0006
SFTON P0349
REFP 3 C00103 BC00103
CALL JOB:SEARCH-R1
SET P0349 P0006
SFTON P0349
SFTOF
MOVL C00104 BC00104 V=500.0 PL=0
'------------------------
'W251A
'------------------------
MOVL C00105 BC00105 V=333.3 PL=0
REFP 3 C00106 BC00106
CALL JOB:SEARCH-R1
IMOV P0058 V=16.7
SET P0350 P0006
SFTON P0350
REFP 3 C00107 BC00107
CALL JOB:SEARCH-R1
SET P0350 P0006
SFTON P0350
MOVL C00108 BC00108 V=500.0 PL=0
SFTOF
'------------------------
'W254A P
'------------------------
MOVJ C00109 BC00109 VJ=30.00
MOVL C00110 BC00110 V=333.3 PL=0
REFP 3 C00111 BC00111
CALL JOB:SEARCH-R1
IMOV P0058 V=16.7
SET P0351 P0006
SFTON P0351
REFP 3 C00112 BC00112
CALL JOB:SEARCH-R1
SET P0351 P0006
SFTON P0351
MOVL C00113 BC00113 V=500.0 PL=0
SFTOF
'------------------------
'W254A L
'------------------------
MOVJ C00114 BC00114 VJ=30.00
MOVL C00115 BC00115 V=333.3 PL=0
REFP 3 C00116 BC00116
CALL JOB:SEARCH-R1
IMOV P0058 V=16.7
SET P0352 P0006
SFTON P0352
REFP 3 C00117 BC00117
CALL JOB:SEARCH-R1
SET P0352 P0006
SFTON P0352
MOVL C00118 BC00118 V=500.0 PL=0
SFTOF
'------------------------
'W250A P
'------------------------
MOVJ C00119 BC00119 VJ=30.00
MOVL C00120 BC00120 V=333.3 PL=0
REFP 3 C00121 BC00121
CALL JOB:SEARCH-R1
IMOV P0058 V=16.7
SET P0353 P0006
SFTON P0353
REFP 3 C00122 BC00122
CALL JOB:SEARCH-R1
SET P0353 P0006
SFTON P0353
MOVL C00123 BC00123 V=500.0 PL=0
SFTOF
'------------------------
'W250A L
'------------------------
MOVJ C00124 BC00124 VJ=30.00
MOVL C00125 BC00125 V=333.3 PL=0
REFP 3 C00126 BC00126
CALL JOB:SEARCH-R1
IMOV P0058 V=16.7
SET P0354 P0006
SFTON P0354
REFP 3 C00127 BC00127
CALL JOB:SEARCH-R1
SET P0354 P0006
SFTON P0354
MOVL C00128 BC00128 V=500.0 PL=0
SFTOF
'------------------------
'W253A P
'------------------------
MOVJ C00129 BC00129 VJ=30.00
MOVL C00130 BC00130 V=333.3 PL=0
REFP 3 C00131 BC00131
CALL JOB:SEARCH-R1
IMOV P0058 V=16.7
SET P0355 P0006
SFTON P0355
REFP 3 C00132 BC00132
CALL JOB:SEARCH-R1
SET P0355 P0006
SFTON P0355
MOVL C00133 BC00133 V=333.3 PL=0
SFTOF
'------------------------
'W253A L
'------------------------
MOVJ C00134 BC00134 VJ=30.00
MOVL C00135 BC00135 V=333.3 PL=0
REFP 3 C00136 BC00136
CALL JOB:SEARCH-R1
IMOV P0058 V=16.7
SET P0356 P0006
SFTON P0356
REFP 3 C00137 BC00137
CALL JOB:SEARCH-R1
SET P0356 P0006
SFTON P0356
MOVL C00138 BC00138 V=500.0 PL=0
SFTOF
'------------------------
'W256A P
'------------------------
MOVJ C00139 BC00139 VJ=30.00
MOVL C00140 BC00140 V=333.3 PL=0
REFP 3 C00141 BC00141
CALL JOB:SEARCH-R1
IMOV P0058 V=16.7
SET P0357 P0006
SFTON P0357
REFP 3 C00142 BC00142
CALL JOB:SEARCH-R1
SET P0357 P0006
SFTON P0357
MOVL C00143 BC00143 V=500.0 PL=0
SFTOF
'------------------------
'W256A L
'------------------------
MOVJ C00144 BC00144 VJ=30.00
MOVL C00145 BC00145 V=333.3 PL=0
REFP 3 C00146 BC00146
CALL JOB:SEARCH-R1
IMOV P0058 V=16.7
SET P0358 P0006
SFTON P0358
REFP 3 C00147 BC00147
CALL JOB:SEARCH-R1
SET P0358 P0006
SFTON P0358
MOVL C00148 BC00148 V=500.0 PL=0
SFTOF
'------------------------
'W252A P
'------------------------
MOVL C00149 BC00149 V=500.0
MOVL C00150 BC00150 V=333.3 PL=0
REFP 3 C00151 BC00151
CALL JOB:SEARCH-R1
IMOV P0058 V=16.7
SET P0359 P0006
SFTON P0359
REFP 3 C00152 BC00152
CALL JOB:SEARCH-R1
SET P0359 P0006
SFTON P0359
MOVL C00153 BC00153 V=333.3 PL=0
SFTOF
'------------------------
'W252A L
'------------------------
MOVL C00154 BC00154 V=500.0
MOVL C00155 BC00155 V=333.3 PL=0
REFP 3 C00156 BC00156
CALL JOB:SEARCH-R1
IMOV P0058 V=16.7
SET P0360 P0006
SFTON P0360
REFP 3 C00157 BC00157
CALL JOB:SEARCH-R1
SET P0360 P0006
SFTON P0360
MOVL C00158 BC00158 V=500.0 PL=0
SFTOF
'------------------------
'W255A
'------------------------
MOVL C00159 BC00159 V=500.0
MOVL C00160 BC00160 V=333.3 PL=0
REFP 3 C00161 BC00161
CALL JOB:SEARCH-R1
IMOV P0058 V=16.7
SET P0361 P0006
SFTON P0361
REFP 3 C00162 BC00162
CALL JOB:SEARCH-R1
SET P0361 P0006
SFTON P0361
MOVL C00163 BC00163 V=500.0 PL=0
SFTOF
'------------------------
'W255A
'------------------------
MOVL C00164 BC00164 V=500.0
MOVL C00165 BC00165 V=333.3 PL=0
REFP 3 C00166 BC00166
CALL JOB:SEARCH-R1
IMOV P0058 V=16.7
SET P0362 P0006
SFTON P0362
REFP 3 C00167 BC00167
CALL JOB:SEARCH-R1
SET P0362 P0006
SFTON P0362
MOVL C00168 BC00168 V=500.0 PL=0
SFTOF
MOVL C00169 BC00169 V=500.0
MOVJ C00170 BC00170 VJ=50.00
MOVJ C00171 BC00171 VJ=50.00
MOVJ C00172 BC00172 VJ=50.00
COMM MOVJ C00173 BC00173 VJ=30.00
COMM MOVJ C00174 BC00174 VJ=30.00
COMM MOVJ C00175 BC00175 VJ=30.00
COMM MOVJ C00176 BC00176 VJ=50.00
COMM 'COMMENT
COMM MOVJ C00177 BC00177 VJ=50.00
COMM MOVJ C00178 BC00178 VJ=30.00
COMM GETE D040 P0400 (1)
COMM GETE D041 P0400 (2)
COMM GETE D042 P0400 (3)
COMM SETE P0401 (1) D040
COMM SETE P0401 (2) D041
COMM SETE P0401 (3) D042
COMM GETE D040 P0400 (1)
COMM GETE D041 P0400 (2)
COMM GETE D042 P0400 (3)
COMM SETE P0402 (1) D040
COMM SETE P0402 (2) D041
COMM SETE P0402 (3) D042
COMM MOVL C00179 BC00179 V=333.3
COMM MOVL C00180 BC00180 V=333.3
COMM MOVL C00181 BC00181 V=333.3
COMM MOVL C00182 BC00182 V=333.3
COMM '------------------------
COMM 'W61.5
COMM '------------------------
COMM MOVL C00183 BC00183 V=66.7 PL=0
COMM REFP 3 C00184 BC00184
COMM CALL JOB:SEARCH-R1
COMM SET P0401 P0006
COMM SFTON P0401
COMM MOVL C00185 BC00185 V=66.7 PL=0
COMM REFP 3 C00186 BC00186
COMM CALL JOB:SEARCH-R1
COMM SET P0401 P0006
COMM SFTON P0401
COMM MOVL C00187 BC00187 V=66.7 PL=0
COMM SFTOF
COMM MOVL C00188 BC00188 V=333.3
COMM MOVL C00189 BC00189 V=333.3
COMM '------------------------
COMM 'W61.7
COMM '------------------------
COMM MOVL C00190 BC00190 V=333.3
COMM MOVL C00191 BC00191 V=66.7 PL=0
COMM REFP 3 C00192 BC00192
COMM CALL JOB:SEARCH-R1
COMM SET P0402 P0006
COMM SFTON P0402
COMM MOVL C00193 BC00193 V=66.7 PL=0
COMM REFP 3 C00194 BC00194
COMM CALL JOB:SEARCH-R1
COMM SET P0402 P0006
COMM SFTON P0402
COMM MOVL C00195 BC00195 V=66.7 PL=0
COMM SFTOF
COMM '------------------------
COMM 'W61.10
COMM '------------------------
COMM MOVL C00196 BC00196 V=500.0
COMM MOVL C00197 BC00197 V=166.7 PL=0
COMM REFP 3 C00198 BC00198
COMM CALL JOB:SEARCH-R1
COMM SET P0403 P0006
COMM SFTON P0403
COMM MOVL C00199 BC00199 V=166.7 PL=0
COMM REFP 3 C00200 BC00200
COMM CALL JOB:SEARCH-R1
COMM SET P0403 P0006
COMM SFTON P0403
COMM MOVL C00201 BC00201 V=500.0 PL=0
COMM SFTOF
COMM '------------------------
COMM 'W61.12
COMM '------------------------
COMM MOVL C00202 BC00202 V=500.0
COMM MOVL C00203 BC00203 V=166.7 PL=0
COMM REFP 3 C00204 BC00204
COMM CALL JOB:SEARCH-R1
COMM SET P0404 P0006
COMM SFTON P0404
COMM MOVL C00205 BC00205 V=166.7 PL=0
COMM REFP 3 C00206 BC00206
COMM CALL JOB:SEARCH-R1
COMM SET P0404 P0006
COMM SFTON P0404
COMM MOVL C00207 BC00207 V=500.0 PL=0
COMM SFTOF
COMM '------------------------
COMM 'W61.15
COMM '------------------------
COMM MOVL C00208 BC00208 V=500.0
COMM MOVL C00209 BC00209 V=166.7 PL=0
COMM REFP 3 C00210 BC00210
COMM CALL JOB:SEARCH-R1
COMM SET P0405 P0006
COMM SFTON P0405
COMM MOVL C00211 BC00211 V=166.7 PL=0
COMM REFP 3 C00212 BC00212
COMM CALL JOB:SEARCH-R1
COMM SET P0405 P0006
COMM SFTON P0405
COMM MOVL C00213 BC00213 V=500.0 PL=0
COMM SFTOF
COMM MOVL C00214 BC00214 V=500.0
COMM SFTOF
COMM GETE D040 P0405 (1)
COMM GETE D041 P0405 (2)
COMM GETE D042 P0405 (3)
COMM SETE P0406 (1) D040
COMM SETE P0406 (2) D041
COMM SETE P0406 (3) D042
COMM '------------------------
COMM 'W61.17
COMM '------------------------
COMM MOVL C00215 BC00215 V=333.3
COMM MOVL C00216 BC00216 V=66.7 PL=0
COMM REFP 3 C00217 BC00217
COMM CALL JOB:SEARCH-R1
COMM SET P0406 P0006
COMM SFTON P0406
COMM MOVL C00218 BC00218 V=66.7 PL=0
COMM REFP 3 C00219 BC00219
COMM CALL JOB:SEARCH-R1
COMM SET P0406 P0006
COMM SFTON P0406
COMM MOVL C00220 BC00220 V=66.7 PL=0
COMM SFTOF
COMM MOVL C00221 BC00221 V=333.3
COMM MOVL C00222 BC00222 V=333.3
COMM MOVJ C00223 BC00223 VJ=30.00
COMM MOVJ C00224 BC00224 VJ=50.00
COMM MOVL C00225 BC00225 V=666.7
COMM '------------------------
COMM 'W61.20
COMM '------------------------
COMM MOVL C00226 BC00226 V=500.0
COMM MOVL C00227 BC00227 V=166.7 PL=0
COMM REFP 3 C00228 BC00228
COMM CALL JOB:SEARCH-R1
COMM SET P0407 P0006
COMM SFTON P0407
COMM MOVL C00229 BC00229 V=166.7 PL=0
COMM REFP 3 C00230 BC00230
COMM CALL JOB:SEARCH-R1
COMM SET P0407 P0006
COMM SFTON P0407
COMM MOVL C00231 BC00231 V=500.0 PL=0
COMM SFTOF
COMM '------------------------
COMM 'W61.23
COMM '------------------------
COMM MOVL C00232 BC00232 V=500.0
COMM MOVL C00233 BC00233 V=166.7 PL=0
COMM REFP 3 C00234 BC00234
COMM CALL JOB:SEARCH-R1
COMM SET P0408 P0006
COMM SFTON P0408
COMM MOVL C00235 BC00235 V=166.7 PL=0
COMM REFP 3 C00236 BC00236
COMM CALL JOB:SEARCH-R1
COMM SET P0408 P0006
COMM SFTON P0408
COMM MOVL C00237 BC00237 V=500.0 PL=0
COMM SFTOF
COMM '------------------------
COMM 'W61.25
COMM '------------------------
COMM MOVL C00238 BC00238 V=500.0
COMM MOVL C00239 BC00239 V=166.7 PL=0
COMM REFP 3 C00240 BC00240
COMM CALL JOB:SEARCH-R1
COMM SET P0409 P0006
COMM SFTON P0409
COMM MOVL C00241 BC00241 V=166.7 PL=0
COMM REFP 3 C00242 BC00242
COMM CALL JOB:SEARCH-R1
COMM SET P0409 P0006
COMM SFTON P0409
COMM MOVL C00243 BC00243 V=500.0 PL=0
COMM SFTOF
COMM MOVL C00244 BC00244 V=500.0
COMM MOVL C00245 BC00245 V=500.0
COMM MOVJ C00246 BC00246 VJ=50.00
COMM MOVL C00247 BC00247 V=666.7
COMM GETE D040 P0409 (1)
COMM GETE D041 P0409 (2)
COMM GETE D042 P0409 (3)
COMM SETE P0410 (1) D040
COMM SETE P0410 (2) D041
COMM SETE P0410 (3) D042
COMM '------------------------
COMM 'W61.30
COMM '------------------------
COMM MOVL C00248 BC00248 V=500.0
COMM MOVL C00249 BC00249 V=166.7 PL=0
COMM REFP 3 C00250 BC00250
COMM CALL JOB:SEARCH-R1
COMM SET P0411 P0006
COMM SFTON P0411
COMM MOVL C00251 BC00251 V=166.7 PL=0
COMM REFP 3 C00252 BC00252
COMM CALL JOB:SEARCH-R1
COMM SET P0411 P0006
COMM SFTON P0411
COMM MOVL C00253 BC00253 V=500.0 PL=0
COMM SFTOF
COMM MOVL C00254 BC00254 V=666.7
COMM MOVJ C00255 BC00255 VJ=30.00
MOVJ C00256 BC00256 VJ=50.00
CALL JOB:FRONT_SEARCH_90ST-2_5440
MOVJ C00257 BC00257 VJ=50.00
MOVJ C00258 BC00258 VJ=40.00
MOVJ C00259 BC00259 VJ=30.00
MOVL C00260 BC00260 V=666.7
MOVJ C00261 BC00261 VJ=40.00
'------------------------
'W65.3
'------------------------
SFTON P0300
MOVL C00262 BC00262 V=500.0
MOVL C00263 BC00263 V=333.3 PL=0
MACRO1 MJ#(0) ARGF10
ARCON
MOVL C00264 BC00264 V=10.8
ARCOF
MOVL C00265 BC00265 V=166.7
SFTOF
'------------------------
'W65.5
'------------------------
SFTON P0301
MOVL C00266 BC00266 V=333.3
MOVL C00267 BC00267 V=133.3 PL=0
MACRO1 MJ#(0) ARGF10
ARCON
MOVL C00268 BC00268 V=10.8
ARCOF
MOVL C00269 BC00269 V=166.7
SFTOF
MOVL C00270 BC00270 V=500.0
MOVL C00271 BC00271 V=333.3
MOVJ C00272 BC00272 VJ=25.00
MOVJ C00273 BC00273 VJ=50.00
'::::::::::::::::::::::::::::::::
'::::::::::::::::::::::::::::::::
'::::::::::::::::::::::::::::::::
'::::::::::::::::::::::::::::::::
'::::::::::::::::::::::::::::::::
COMM MOVJ C00274 BC00274 VJ=50.00
COMM MOVJ C00275 BC00275 VJ=50.00
COMM MOVJ C00276 BC00276 VJ=50.00
COMM MOVJ C00277 BC00277 VJ=50.00
COMM MOVJ C00278 BC00278 VJ=20.00
COMM '------------------------
COMM 'W61.3
COMM '------------------------
COMM SFTON P0400
COMM MOVL C00279 BC00279 V=333.3
COMM MOVL C00280 BC00280 V=66.7 PL=0
COMM MACRO1 MJ#(0) ARGF9
COMM ARCOF
COMM SFTOF
COMM 'BELKA PRZEJAZD
COMM MOVJ C00281 BC00281 VJ=25.00
COMM MOVJ C00282 BC00282 VJ=50.00
COMM MOVL C00283 BC00283 V=500.0
COMM MOVL C00284 BC00284 V=500.0
COMM '------------------------
COMM 'W61.5
COMM '------------------------
COMM SFTON P0401
COMM MOVL C00285 BC00285 V=333.3
COMM MOVL C00286 BC00286 V=133.3 PL=0
COMM MACRO1 MJ#(0) ARGF24
COMM ARCON
COMM MOVL C00287 BC00287 V=7.5
COMM ARCOF
COMM MOVL C00288 BC00288 V=250.0
COMM SFTOF
COMM MOVL C00289 BC00289 V=333.3
COMM MOVJ C00290 BC00290 VJ=35.00
COMM MOVJ C00291 BC00291 VJ=50.00
COMM MOVJ C00292 BC00292 VJ=50.00
COMM MOVJ C00293 BC00293 VJ=50.00
MOVJ C00294 BC00294 VJ=50.00
MOVJ C00295 BC00295 VJ=50.00
MOVJ C00296 BC00296 VJ=50.00
'------------------------
'W250A
'------------------------
SFTON P0354
MOVL C00297 BC00297 V=333.3
MOVL C00298 BC00298 V=133.3 PL=0
MACRO1 MJ#(0) ARGF9
ARCON
SFTOF
SFTON P0353
MOVL C00299 BC00299 V=11.7
ARCOF
MOVL C00300 BC00300 V=166.7
SFTOF
MOVJ C00301 BC00301 VJ=50.00
MOVJ C00302 BC00302 VJ=50.00
MOVJ C00303 BC00303 VJ=50.00
MOVJ C00304 BC00304 VJ=50.00
MOVJ C00305 BC00305 VJ=50.00
MOVJ C00306 BC00306 VJ=20.00
MOVJ C00307 BC00307 VJ=10.00
'------------------------
'W65.7
'------------------------
SFTON P0302
'MOTOSIM PULSE LIMIT
MOVL C00308 BC00308 V=500.0
MOVL C00309 BC00309 V=133.3 PL=0
MACRO1 MJ#(0) ARGF10
ARCON
MOVL C00310 BC00310 V=10.8
ARCOF
MOVL C00311 BC00311 V=250.0
SFTOF
'------------------------
'W65.10
'------------------------
SFTON P0303
MOVL C00312 BC00312 V=500.0
MOVL C00313 BC00313 V=166.7 PL=0
ARCON
MOVL C00314 BC00314 V=10.8
ARCOF
MOVL C00315 BC00315 V=166.7
SFTOF
SFTOF
MOVL C00316 BC00316 V=333.3
MOVL C00317 BC00317 V=500.0
MOVJ C00318 BC00318 VJ=50.00
MOVJ C00319 BC00319 VJ=30.00
MOVJ C00320 BC00320 VJ=50.00
MOVJ C00321 BC00321 VJ=50.00
COMM '::::::::::::::::::::::::::::::::
COMM '::::::::::::::::::::::::::::::::
COMM '------------------------
COMM 'W61.7
COMM '------------------------
COMM '::::::::::::::::::::::::::::::::
COMM '::::::::::::::::::::::::::::::::
COMM MOVJ C00322 BC00322 VJ=50.00
COMM MOVJ C00323 BC00323 VJ=35.00
COMM SFTON P0402
COMM MOVL C00324 BC00324 V=333.3
COMM MOVL C00325 BC00325 V=133.3 PL=0
COMM MACRO1 MJ#(0) ARGF24
COMM ARCON
COMM MOVL C00326 BC00326 V=7.5
COMM ARCOF
COMM MOVL C00327 BC00327 V=166.7
COMM SFTOF
COMM MOVL C00328 BC00328 V=500.0
COMM MOVL C00329 BC00329 V=500.0
COMM MOVJ C00330 BC00330 VJ=50.00
COMM '------------------------
COMM 'W61.10
COMM '------------------------
COMM SFTON P0403
COMM MOVL C00331 BC00331 V=333.3
COMM MOVL C00332 BC00332 V=133.3 PL=0
COMM MACRO1 MJ#(0) ARGF24
COMM ARCON
COMM MOVL C00333 BC00333 V=7.5
COMM ARCOF
COMM MOVL C00334 BC00334 V=166.7
COMM SFTOF
COMM MOVL C00335 BC00335 V=333.3
COMM MOVJ C00336 BC00336 VJ=35.00
COMM MOVJ C00337 BC00337 VJ=50.00
COMM MOVJ C00338 BC00338 VJ=50.00
COMM '::::::::::::::::::::::::
COMM '::::::::::::::::::::::::
COMM '::::::::::::::::::::::::
COMM '::::::::::::::::::::::::
COMM '::::::::::::::::::::::::
COMM '::::::::::::::::::::::::
COMM '::::::::::::::::::::::::
MOVJ C00339 BC00339 VJ=50.00
MOVJ C00340 BC00340 VJ=50.00
MOVJ C00341 BC00341 VJ=50.00
'------------------------
'W214A
'------------------------
SFTON P0350
MOVL C00342 BC00342 V=333.3
MOVL C00343 BC00343 V=333.3
MOVL C00344 BC00344 V=133.3 PL=0
MACRO1 MJ#(0) ARGF9
ARCON
SFTOF
SFTON P0349
MOVL C00345 BC00345 V=11.7
MOVL C00346 BC00346 V=11.2
ARCOF
MOVL C00347 BC00347 V=416.7
SFTOF
MOVJ C00348 BC00348 VJ=50.00
MOVJ C00349 BC00349 VJ=50.00
MOVJ C00350 BC00350 VJ=50.00
MOVJ C00351 BC00351 VJ=50.00
MOVJ C00352 BC00352 VJ=50.00
MOVJ C00353 BC00353 VJ=50.00
MOVJ C00354 BC00354 VJ=20.00
'------------------------
'W65.12
'------------------------
SFTON P0304
MOVL C00355 BC00355 V=333.3
MOVL C00356 BC00356 V=133.3 PL=0
MACRO1 MJ#(0) ARGF10
ARCON
MOVL C00357 BC00357 V=10.8
ARCOF
MOVL C00358 BC00358 V=166.7
SFTOF
'------------------------
'W65.15
'------------------------
SFTON P0305
MOVL C00359 BC00359 V=333.3
MOVL C00360 BC00360 V=166.7 PL=0
MACRO1 MJ#(0) ARGF10
ARCON
MOVL C00361 BC00361 V=10.8
ARCOF
MOVL C00362 BC00362 V=166.7
SFTOF
MOVL C00363 BC00363 V=416.7
SFTON P0306
MOVL C00364 BC00364 V=166.7
ARCON
MOVL C00365 BC00365 V=10.8
ARCOF
SFTOF
MOVL C00366 BC00366 V=166.7
MOVL C00367 BC00367 V=333.3
MOVL C00368 BC00368 V=500.0
MOVL C00369 BC00369 V=500.0
MOVJ C00370 BC00370 VJ=50.00
COMM '::::::::::::::::::::::::
COMM '::::::::::::::::::::::::
COMM '::::::::::::::::::::::::
COMM '::::::::::::::::::::::::
COMM '::::::::::::::::::::::::
COMM '::::::::::::::::::::::::
COMM '::::::::::::::::::::::::
COMM MOVJ C00371 BC00371 VJ=50.00
COMM MOVJ C00372 BC00372 VJ=50.00
COMM '::::::::::::::::::::::::::::::::
COMM '::::::::::::::::::::::::::::::::
COMM '------------------------
COMM 'W61.12
COMM '------------------------
COMM '::::::::::::::::::::::::::::::::
COMM '::::::::::::::::::::::::::::::::
COMM SFTON P0404
COMM MOVJ C00373 BC00373 VJ=50.00
COMM MOVL C00374 BC00374 V=333.3
COMM MOVL C00375 BC00375 V=333.3
COMM MOVL C00376 BC00376 V=166.7 PL=0
COMM MACRO1 MJ#(0) ARGF24
COMM ARCON
COMM MOVL C00377 BC00377 V=7.5
COMM ARCOF
COMM MOVL C00378 BC00378 V=166.7
COMM SFTOF
COMM MOVL C00379 BC00379 V=333.3
COMM MOVL C00380 BC00380 V=333.3
COMM '------------------------
COMM 'W61.15
COMM '------------------------
COMM SFTON P0405
COMM MOVL C00381 BC00381 V=333.3
COMM MOVL C00382 BC00382 V=166.7 PL=0
COMM MACRO1 MJ#(0) ARGF24
COMM ARCON
COMM MOVL C00383 BC00383 V=7.5
COMM ARCOF
COMM MOVL C00384 BC00384 V=166.7
COMM SFTOF
COMM MOVJ C00385 BC00385 VJ=50.00
COMM MOVJ C00386 BC00386 VJ=50.00
COMM MOVJ C00387 BC00387 VJ=50.00
COMM '::::::::::::::::::::::::
COMM '::::::::::::::::::::::::
COMM '::::::::::::::::::::::::
COMM '::::::::::::::::::::::::
COMM '::::::::::::::::::::::::
COMM '::::::::::::::::::::::::
COMM '::::::::::::::::::::::::
MOVJ C00388 BC00388 VJ=50.00
MOVJ C00389 BC00389 VJ=50.00
'------------------------
'W252A
'------------------------
SFTON P0359
MOVL C00390 BC00390 V=500.0
MOVL C00391 BC00391 V=166.7 PL=0
MACRO1 MJ#(0) ARGF9
ARCON
SFTOF
SFTON P0358
MOVL C00392 BC00392 V=11.7
ARCOF
MOVL C00393 BC00393 V=250.0
SFTOF
MOVJ C00394 BC00394 VJ=50.00
MOVJ C00395 BC00395 VJ=80.00
COMM MOVJ C00396 BC00396 VJ=50.00
COMM MOVJ C00397 BC00397 VJ=50.00
COMM MOVJ C00398 BC00398 VJ=25.00
COMM MOVL C00399 BC00399 V=333.3
COMM MOVL C00400 BC00400 V=333.3
COMM '------------------------
COMM 'W65.17
COMM '------------------------
COMM SFTON P0306
COMM MOVL C00401 BC00401 V=166.7
COMM MOVL C00402 BC00402 V=166.7 PL=0
COMM MACRO1 MJ#(0) ARGF10
COMM ARCON
COMM MOVL C00403 BC00403 V=10.8
COMM ARCOF
COMM MOVL C00404 BC00404 V=166.7
COMM SFTOF
COMM MOVL C00405 BC00405 V=250.0
COMM MOVL C00406 BC00406 V=250.0
COMM MOVL C00407 BC00407 V=333.3
COMM MOVJ C00408 BC00408 VJ=25.00
COMM '::::::::::::::::::::::::
COMM '::::::::::::::::::::::::
COMM '::::::::::::::::::::::::
COMM '::::::::::::::::::::::::
COMM '::::::::::::::::::::::::
COMM '::::::::::::::::::::::::
COMM '::::::::::::::::::::::::
COMM '::::::::::::::::::::::::::::::::
COMM '::::::::::::::::::::::::::::::::
COMM '------------------------
COMM 'W61.17
COMM '------------------------
COMM '::::::::::::::::::::::::::::::::
COMM '::::::::::::::::::::::::::::::::
COMM SFTON P0406
COMM MOVJ C00409 BC00409 VJ=10.00
COMM MOVL C00410 BC00410 V=150.0
COMM MOVL C00411 BC00411 V=66.7 PL=0
COMM MACRO1 MJ#(0) ARGF24
COMM ARCON
COMM MOVL C00412 BC00412 V=6.7
COMM ARCOF
COMM MOVL C00413 BC00413 V=83.3
COMM SFTOF
'------------------------
'W253A
'------------------------
MOVJ C00414 BC00414 VJ=50.00
SFTON P0356
MOVL C00415 BC00415 V=333.3
MOVL C00416 BC00416 V=333.3
MOVL C00417 BC00417 V=166.7 PL=0
MACRO1 MJ#(0) ARGF9
ARCON
SFTOF
SFTON P0355
MOVL C00418 BC00418 V=11.7
ARCOF
MOVL C00419 BC00419 V=250.0
SFTOF
MOVJ C00420 BC00420 VJ=50.00
MOVJ C00421 BC00421 VJ=50.00
MOVJ C00422 BC00422 VJ=80.00
MOVJ C00423 BC00423 VJ=80.00
MOVJ C00424 BC00424 VJ=50.00
COMM MOVJ C00425 BC00425 VJ=50.00
COMM MOVJ C00426 BC00426 VJ=50.00
COMM MOVJ C00427 BC00427 VJ=30.00
COMM '------------------------
COMM 'W65.20
COMM '------------------------
COMM SFTON P0307
COMM MOVL C00428 BC00428 V=333.3
COMM MOVL C00429 BC00429 V=166.7
COMM MOVL C00430 BC00430 V=166.7 PL=0
COMM MACRO1 MJ#(0) ARGF10
COMM ARCON
COMM MOVL C00431 BC00431 V=10.8
COMM ARCOF
COMM MOVL C00432 BC00432 V=250.0
COMM SFTOF
COMM MOVL C00433 BC00433 V=333.3
COMM MOVL C00434 BC00434 V=333.3
COMM MOVL C00435 BC00435 V=333.3
COMM MOVJ C00436 BC00436 VJ=50.00
COMM MOVJ C00437 BC00437 VJ=50.00
COMM MOVJ C00438 BC00438 VJ=50.00
COMM MOVJ C00439 BC00439 VJ=50.00
COMM '::::::::::::::::::::::::
COMM '::::::::::::::::::::::::
COMM '::::::::::::::::::::::::
COMM '::::::::::::::::::::::::
COMM '::::::::::::::::::::::::
COMM '::::::::::::::::::::::::
COMM '::::::::::::::::::::::::
COMM MOVJ C00440 BC00440 VJ=80.00
COMM MOVJ C00441 BC00441 VJ=50.00
COMM MOVJ C00442 BC00442 VJ=50.00
COMM '::::::::::::::::::::::::::::::::
COMM '::::::::::::::::::::::::::::::::
COMM '------------------------
COMM 'W61.20
COMM '------------------------
COMM '::::::::::::::::::::::::::::::::
COMM '::::::::::::::::::::::::::::::::
COMM SFTON P0407
COMM MOVL C00443 BC00443 V=333.3
COMM MOVL C00444 BC00444 V=166.7
COMM MOVL C00445 BC00445 V=133.3 PL=0
COMM MACRO1 MJ#(0) ARGF24
COMM ARCON
COMM MOVL C00446 BC00446 V=7.5
COMM ARCOF
COMM MOVL C00447 BC00447 V=166.7
COMM SFTOF
COMM SFTON P0407
COMM MOVL C00448 BC00448 V=166.7
COMM MOVL C00449 BC00449 V=133.3 PL=0
COMM MACRO1 MJ#(0) ARGF24
COMM ARCON
COMM MOVL C00450 BC00450 V=7.5
COMM ARCOF
COMM MOVL C00451 BC00451 V=166.7
COMM SFTOF
COMM '::::::::::::::::::::::::
COMM '::::::::::::::::::::::::
COMM '::::::::::::::::::::::::
COMM '::::::::::::::::::::::::
COMM '::::::::::::::::::::::::
COMM MOVJ C00452 BC00452 VJ=50.00
COMM MOVJ C00453 BC00453 VJ=50.00
COMM MOVJ C00454 BC00454 VJ=50.00
COMM MOVJ C00455 BC00455 VJ=50.00
COMM '------------------------
COMM 'W254A
COMM '------------------------
MOVJ C00456 BC00456 VJ=50.00
MOVJ C00457 BC00457 VJ=50.00
SFTON P0352
MOVL C00458 BC00458 V=500.0
MOVL C00459 BC00459 V=500.0
MOVL C00460 BC00460 V=166.7 PL=0
MACRO1 MJ#(0) ARGF9
ARCON
SFTOF
SFTON P0351
MOVL C00461 BC00461 V=11.7
ARCOF
MOVL C00462 BC00462 V=333.3
SFTOF
COMM MOVJ C00463 BC00463 VJ=80.00
COMM MOVJ C00464 BC00464 VJ=80.00
COMM MOVJ C00465 BC00465 VJ=80.00
COMM MOVJ C00466 BC00466 VJ=80.00
COMM MOVJ C00467 BC00467 VJ=50.00
MOVJ C00468 BC00468 VJ=50.00
MOVJ C00469 BC00469 VJ=50.00
MOVL C00470 BC00470 V=500.0
'------------------------
'W65.23
'------------------------
SFTON P0308
MOVL C00471 BC00471 V=333.3
MOVL C00472 BC00472 V=166.7
MOVL C00473 BC00473 V=133.3 PL=0
MACRO1 MJ#(0) ARGF10
ARCON
MOVL C00474 BC00474 V=10.8
ARCOF
MOVL C00475 BC00475 V=166.7
SFTOF
'------------------------
'W65.25
'------------------------
SFTON P0309
MOVL C00476 BC00476 V=500.0
MOVL C00477 BC00477 V=133.3 PL=0
ARCON
MOVL C00478 BC00478 V=10.8
ARCOF
MOVL C00479 BC00479 V=166.7
SFTOF
MOVL C00480 BC00480 V=333.3
SFTON P0310
MOVL C00481 BC00481 V=166.7
ARCON
MOVL C00482 BC00482 V=10.8
ARCOF
SFTOF
MOVL C00483 BC00483 V=166.7
MOVL C00484 BC00484 V=500.0
MOVL C00485 BC00485 V=333.3
MOVL C00486 BC00486 V=500.0
MOVL C00487 BC00487 V=333.3
MOVJ C00488 BC00488 VJ=50.00
MOVJ C00489 BC00489 VJ=50.00
MOVJ C00490 BC00490 VJ=50.00
MOVJ C00491 BC00491 VJ=80.00
COMM '::::::::::::::::::::::::
COMM '::::::::::::::::::::::::
COMM '::::::::::::::::::::::::
COMM '::::::::::::::::::::::::
COMM '::::::::::::::::::::::::
COMM '::::::::::::::::::::::::
COMM '::::::::::::::::::::::::
COMM MOVJ C00492 BC00492 VJ=80.00
COMM MOVJ C00493 BC00493 VJ=80.00
COMM MOVJ C00494 BC00494 VJ=50.00
COMM MOVJ C00495 BC00495 VJ=50.00
COMM '::::::::::::::::::::::::::::::::
COMM '::::::::::::::::::::::::::::::::
COMM '------------------------
COMM 'W61.23
COMM '------------------------
COMM '::::::::::::::::::::::::::::::::
COMM '::::::::::::::::::::::::::::::::
COMM SFTON P0408
COMM MOVL C00496 BC00496 V=333.3
COMM MOVL C00497 BC00497 V=166.7
COMM MOVL C00498 BC00498 V=133.3 PL=0
COMM MACRO1 MJ#(0) ARGF24
COMM ARCON
COMM MOVL C00499 BC00499 V=7.5
COMM ARCOF
COMM MOVL C00500 BC00500 V=83.3
COMM SFTOF
COMM '------------------------
COMM 'W61.25
COMM '------------------------
COMM SFTON P0409
COMM MOVL C00501 BC00501 V=333.3
COMM MOVL C00502 BC00502 V=150.0
COMM MOVL C00503 BC00503 V=133.3 PL=0
COMM MACRO1 MJ#(0) ARGF24
COMM ARCON
COMM MOVL C00504 BC00504 V=7.5
COMM ARCOF
COMM MOVL C00505 BC00505 V=166.7
COMM SFTOF
COMM '::::::::::::::::::::::::
COMM '::::::::::::::::::::::::
COMM '::::::::::::::::::::::::
COMM '::::::::::::::::::::::::
COMM '::::::::::::::::::::::::
COMM MOVL C00506 BC00506 V=333.3
COMM MOVJ C00507 BC00507 VJ=50.00
COMM MOVJ C00508 BC00508 VJ=50.00
COMM MOVJ C00509 BC00509 VJ=50.00
COMM MOVJ C00510 BC00510 VJ=50.00
MOVJ C00511 BC00511 VJ=80.00
'------------------------
'W255A
MOVL C00512 BC00512 V=500.0
MOVL C00513 BC00513 V=333.3
SFTON P0361
MOVL C00514 BC00514 V=133.3 PL=0
MACRO1 MJ#(0) ARGF9
ARCON
SFTON P0362
MOVL C00515 BC00515 V=11.7
MOVL C00516 BC00516 V=11.2
ARCOF
MOVL C00517 BC00517 V=250.0
SFTOF
MOVL C00518 BC00518 V=333.3
MOVL C00519 BC00519 V=333.3
MOVL C00520 BC00520 V=500.0
MOVJ C00521 BC00521 VJ=50.00
MOVJ C00522 BC00522 VJ=50.00
MOVJ C00523 BC00523 VJ=80.00
MOVJ C00524 BC00524 VJ=50.00
MOVJ C00525 BC00525 VJ=50.00
MOVL C00526 BC00526 V=333.3
'------------------------
'W31.28
'------------------------
COMM SFTON P0310
COMM MOVL C00527 BC00527 V=333.3
COMM MOVL C00528 BC00528 V=333.3
COMM MOVL C00529 BC00529 V=166.7
COMM MOVL C00530 BC00530 V=66.7 PL=0
COMM MACRO1 MJ#(0) ARGF24
COMM ARCON
COMM MOVL C00531 BC00531 V=8.3
COMM ARCOF
COMM MOVL C00532 BC00532 V=83.3
COMM SFTOF
COMM '------------------------
COMM 'W31.30
'------------------------
SFTON P0311
MOVL C00533 BC00533 V=333.3
MOVL C00534 BC00534 V=133.3 PL=0
MACRO1 MJ#(0) ARGF10
ARCON
MOVL C00535 BC00535 V=10.8
ARCOF
SFTOF
MOVL C00536 BC00536 V=166.7
MOVL C00537 BC00537 V=333.3
SFTON P0312
MOVL C00538 BC00538 V=166.7
ARCON
MOVL C00539 BC00539 V=10.8
ARCOF
MOVL C00540 BC00540 V=166.7
MOVL C00541 BC00541 V=166.7
ARCON
MOVL C00542 BC00542 V=10.8
ARCOF
SFTOF
MOVL C00543 BC00543 V=166.7
MOVL C00544 BC00544 V=333.3
SFTOF
MOVL C00545 BC00545 V=500.0
MOVL C00546 BC00546 V=333.3
'::::::::::::::::::::::::
'::::::::::::::::::::::::
'::::::::::::::::::::::::
'::::::::::::::::::::::::
'::::::::::::::::::::::::
'::::::::::::::::::::::::
'::::::::::::::::::::::::
MOVJ C00547 BC00547 VJ=50.00 PL=0
COMM MOVJ C00548 BC00548 VJ=50.00
COMM MOVJ C00549 BC00549 VJ=50.00
COMM '::::::::::::::::::::::::::::::::
COMM '::::::::::::::::::::::::::::::::
COMM '------------------------
COMM 'W61.30
COMM '------------------------
COMM '::::::::::::::::::::::::::::::::
COMM '::::::::::::::::::::::::::::::::
COMM SFTON P0411
COMM MOVL C00550 BC00550 V=333.3
COMM MOVL C00551 BC00551 V=133.3 PL=0
COMM MACRO1 MJ#(0) ARGF24
COMM ARCON
COMM MOVL C00552 BC00552 V=7.5
COMM ARCOF
COMM MOVL C00553 BC00553 V=166.7
COMM SFTOF
COMM MOVL C00554 BC00554 V=500.0
COMM MOVJ C00555 BC00555 VJ=50.00
COMM MOVJ C00556 BC00556 VJ=50.00
COMM MOVJ C00557 BC00557 VJ=50.00
COMM MOVJ C00558 BC00558 VJ=80.00
COMM MOVJ C00559 BC00559 VJ=80.00
COMM '------------------------
COMM 'W256A
COMM '------------------------
MOVJ C00560 BC00560 VJ=80.00
MOVJ C00561 BC00561 VJ=80.00
SFTON P0358
MOVL C00562 BC00562 V=333.3
MOVL C00563 BC00563 V=250.0
MOVL C00564 BC00564 V=166.7 PL=0
MACRO1 MJ#(0) ARGF9
ARCON
SFTOF
SFTON P0357
MOVL C00565 BC00565 V=11.7
ARCOF
MOVL C00566 BC00566 V=333.3
SFTOF
MOVJ C00567 BC00567 VJ=50.00
MOVJ C00568 BC00568 VJ=50.00
MOVJ C00569 BC00569 VJ=80.00
CALL JOB:FRONT_WELD_90ST-2_5440
CALL JOB:MOVE_OUT_OF_TUNNEL
END
